Fanuc KAREL source: kb00015.KL

-- PROVISIONAL review KL for V770-1; original PC SHA256 bd461ddf3c6f4d856ce02dbeaa132ebedfbabd3c9f639223f0a033ecc2a6ec36
-- Incomplete behavior may be omitted. Consult companion uncertainty JSON. Do not deploy.
PROGRAM KB00015
%NOLOCKGROUP
BEGIN
  -- UNRESOLVED_PC offsets 5-14; opcodes 3F,75
  -- UNRESOLVED_PC offsets 19-26; opcodes 9D,23
  -- UNRESOLVED_PC offsets 31-49; opcodes 27,22,2A,22,31
  -- UNRESOLVED_PC offsets 54-58; opcodes 7F
END KB00015
